{attribute 'qualified_only'}
VAR_GLOBAL
	nErrorCodeOKId:UDINT:=0;
	nErrorCodeOKStr:STRING:='NO ERROR';
	nErrorNoLatchId:UDINT:=1000;
	sErrorNoLatchStr:STRING:='NO LATCH FROM DRIVE';
END_VAR

(* stored: Version 1.1.0.1, ProductVersion 3.1.4022.6
   GVL GVL_ErrorCodes: Id {2a5675cd-f9a5-4b29-8d57-a071f0a61152} *)
